ADAPTER BoolAdp (* Adapter Interface *)
  (* Standard: 61499-1 *)
  (* Version 0.0, 7/15/2023, vv263, nxtControl GmBH *)
  PACKAGE Main;
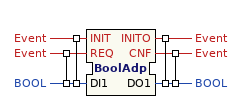
  EVENT_INPUT
    INIT WITH DI1;
    REQ WITH DI1; (* Request from Socket *)
  END_EVENT
  EVENT_OUTPUT
    INITO WITH DO1;
    CNF WITH DO1; (* Confirmation from Plug *)
  END_EVENT
  VAR_INPUT
    DI1 : BOOL; (* Request Data from Socket *)
  END_VAR
  VAR_OUTPUT
    DO1 : BOOL; (* Confirmation Data from Plug *)
  END_VAR
  SERVICE SOCKET/PLUG
    SEQUENCE request_confirm
      SOCKET.REQ(DI1) -> PLUG.REQ(DI1);
      PLUG.CNF(DO1) -> SOCKET.CNF(DO1);
    END_SEQUENCE
    SEQUENCE indication_response
      PLUG.IND(INDD) -> SOCKET.IND(INDD);
      SOCKET.RSP(RSPD) -> PLUG.RSP(RSPD);
    END_SEQUENCE
  END_SERVICE
END_ADAPTER
